// TIA Portal V17 export
// export: Created 2025-03-07T09:19:17.049059Z, ExportSetting WithDefaults, DisplayName Totally Integrated Automation Portal, DisplayVersion V17 Update 8, DisplayName TIA Portal Openness, DisplayVersion V17 Update 8, DisplayName TIA Portal Version Control Interface, DisplayVersion V17, DisplayName SINAMICS Startdrive Advanced, DisplayVersion V17 SP2, DisplayName SINAMICS Startdrive G110M, G120, G120C, G120D, G120P, G115D, DisplayVersion V17 SP2, DisplayName SINAMICS Startdrive G130, G150, S120, S150, SINAMICS MV, S210, DisplayVersion V17 SP2, DisplayName STEP 7 Professional, DisplayVersion V17 Update 8, DisplayName SINUMERIK ONE STEP 7 Toolbox, DisplayVersion V17 Update 12, DisplayName SINUMERIK 840D sl STEP 7 Toolbox, DisplayVersion V17 Update 12, DisplayName STEP 7 Safety, DisplayVersion V17 Update 6, DisplayName WinCC Advanced, DisplayVersion V17 Update 8
DATA_BLOCK "DB7235_VARIABLE_LAYOUT"   // DB7235
{ S7_Optimized_Access := 'FALSE'; DB_Accessible_From_OPC_UA := 'FALSE' }
AUTHOR : ETXETAR
VERSION : 1.0
// stored: AutoNumber false, DBAccessibleFromOPCUA false, DBAccessibleFromWebserver true, IsOnlyStoredInLoadMemory false, IsWriteProtectedInAS false
   VAR RETAIN
      OVERVIEW { S7_SetPoint := 'True'} : "LAYOUT";
      MAGAZINE_01L { S7_SetPoint := 'True'} : "LAYOUT";
      NC_MANUAL { S7_SetPoint := 'True'} : "LAYOUT";
      ETXETAR { S7_SetPoint := 'True'} : "LAYOUT";
      PART_STATUS_UNIT_01 { S7_SetPoint := 'True'} : "LAYOUT";
      QUALITY { S7_SetPoint := 'True'} : "LAYOUT";
      PART_STATUS_UNIT_02 { S7_SetPoint := 'True'} : "LAYOUT";
      PART_ID_UNIT_01 { S7_SetPoint := 'True'} : "LAYOUT";
      PART_ID_UNIT_02 { S7_SetPoint := 'True'} : "LAYOUT";
      U01_PC_STATUS { S7_SetPoint := 'True'} : "LAYOUT";
      U02_PC_STATUS { S7_SetPoint := 'True'} : "LAYOUT";
      U03_PC_STATUS { S7_SetPoint := 'True'} : "LAYOUT";
   END_VAR
BEGIN
END_DATA_BLOCK
